# EPICS autosave request: support/optics/2-6-1/opticsApp/Db/orient_xtals_1_settings.req
$(P)orient$(O):xtal_$(N).STR1
$(P)orient$(O):xtal_$(N).DO2
$(P)orient$(O):xtal_$(N).DO3
$(P)orient$(O):xtal_$(N).DO4
$(P)orient$(O):xtal_$(N).DO5
$(P)orient$(O):xtal_$(N).DO6
$(P)orient$(O):xtal_$(N).DO7
$(P)orient$(O):xtal_$(N).DO8
